TEXTLIST TL_E_MESSAGETYPE
  0 = 'eMessageEmpty'
  1 = 'eMessageError'
  2 = 'eMessageWarning'
  3 = 'eMessageInfo'
  4 = 'eMessageVerbose'
   = ''
END_TEXTLIST

(* stored: Version 1.1.0.1
   TextList TL_E_MESSAGETYPE: Id {5d8a55d8-119a-4fab-9c8a-77a3cf1859ba} *)
